PROGRAM MAIN
VAR
END_VAR

END_PROGRAM

(* stored: Version 1.1.0.1
   POU MAIN: Id {e21ee7d8-4416-4723-ab03-ecbd06dca00d} *)
